// TIA Portal V19 export
DATA_BLOCK "ControlNodes"   // DB154
// stored: MemoryReserve 100, Namespace Unit.Em0
   VAR
      em { ExternalWritable := 'False'} : "LAF_typeEmControlNode";
      fuses { ExternalWritable := 'False'} : Struct
         controlVoltage24VOK : Bool;   // TRUE: No Fault
         driveVoltage24OK : Bool;   // TRUE: No Fault
         robotVoltage24VOK : Bool;   // TRUE: No Fault
         "powerSupply 230VDrivesOK" : Bool;   // TRUE: No Fault
         powerSupply230VRobotOK : Bool;   // TRUE: No Fault
         powerSupply230VIpcOk : Bool;   // TRUE: No Fault
         powerSupply230VCompressorOK : Bool;   // TRUE: No Fault
      END_STRUCT;
      airOK { ExternalWritable := 'False'} : Bool;   // Compressed air OK
   END_VAR
BEGIN
   em.status.enabled := true;
END_DATA_BLOCK
